// Mitsubishi GX Works2 project: 0708-mov들   PLC: Q02/Q02H

PROGRAM MAIN
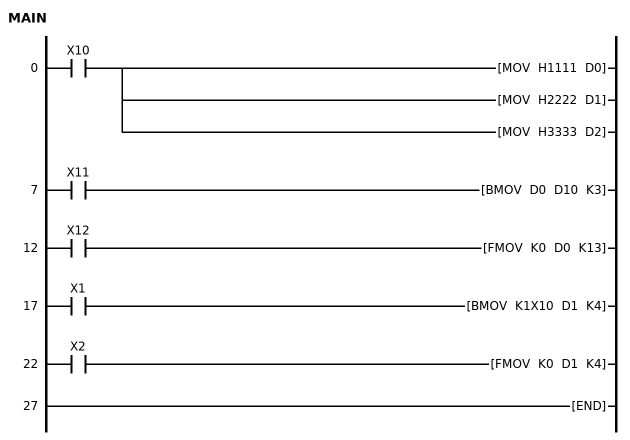
0     LD      X10
      MOV     H1111 D0
      MOV     H2222 D1
      MOV     H3333 D2
7     LD      X11
      BMOV    D0 D10 K3
12    LD      X12
      FMOV    K0 D0 K13
17    LD      X1
      BMOV    K1X10 D1 K4
22    LD      X2
      FMOV    K0 D1 K4
27    END
END_PROGRAM
